FUNCTION_BLOCK SubTank (* Basic Function Block Type *)
  (* Standard: 61499-2 *)
  (* Version 0.0, 2019-06-19, 4DIAC-IDE, 4DIAC-Consortium *)
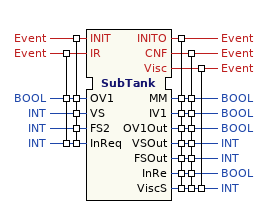
  EVENT_INPUT
    INIT WITH OV1, VS, FS2, InReq; (* Initialization Request *)
    IR WITH OV1, InReq; (* In Flow Request *)
  END_EVENT
  EVENT_OUTPUT
    INITO WITH MM, IV1, ViscS, OV1Out, VSOut, FSOut, InRe; (* Initialization Confirm *)
    CNF WITH MM, IV1, ViscS, OV1Out, VSOut, FSOut, InRe; (* Execution Confirmation *)
    Visc WITH ViscS;
  END_EVENT
  VAR_INPUT
    OV1 : BOOL; (* Outlet Valve *)
    VS : INT; (* Viscosity Sensor *)
    FS2 : INT; (* Fluid Level Sensor *)
    InReq : INT; (* Inlet Request *)
  END_VAR
  VAR_OUTPUT
    MM : BOOL; (* Mixer Motor *)
    IV1 : BOOL; (* Inlet Valve *)
    OV1Out : BOOL;
    VSOut : INT;
    FSOut : INT;
    InRe : BOOL;
    ViscS : INT; (* Viscosity Status *)
  END_VAR
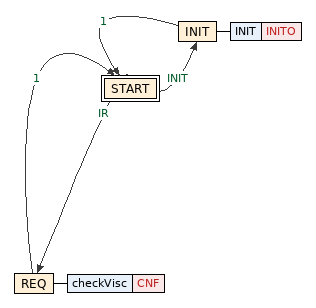
  EC_STATES
    START; (* Initial State *)
    INIT : INIT -> INITO; (* Initialization *)
    REQ : checkVisc -> CNF; (* Normal execution *)
  END_STATES
  EC_TRANSITIONS
    START TO INIT := INIT;
    INIT TO START := 1;
    START TO REQ := IR;
    REQ TO START := 1;
  END_TRANSITIONS
  ALGORITHM INIT IN ST: (* Initialization algorithm *)

  END_ALGORITHM
  ALGORITHM checkVisc IN ST: (* Normally executed algorithm *)
IF VS < 32 THEN
	ViscS := 1;
ELSE
	ViscS := 0;
END_IF;
  END_ALGORITHM
END_FUNCTION_BLOCK
